// TIA Portal project "práctica 20_ comuniacion de plcs" (V15)

(* hardware
DEVICE "S7-1200 station_2"  S7-1200 Station
   slot 0: "Rack_0"  S7-1200 Rack  Rack  V1.0
   slot 1: "PLC_2"  CPU 1214C AC/DC/Rly  6ES7 214-1BG40-0XB0  V4.2
DEVICE "S7-1200 station_1"  S7-1200 Station
   slot 0: "Rack_0"  S7-1200 Rack  Rack  V1.0
   slot 1: "PLC_1"  CPU 1214C AC/DC/Rly  6ES7 214-1BG40-0XB0  V4.2
*)

// ===== PLC "PLC_1"  CPU 1214C AC/DC/Rly =====

VAR_GLOBAL   // PLC tag table "Tabla de variables estándar"
   "System_Byte" AT %MB253 : Byte;
   "FirstScan" AT %M253.0 : Bool;
   "DiagStatusUpdate" AT %M253.1 : Bool;
   "AlwaysTRUE" AT %M253.2 : Bool;
   "AlwaysFALSE" AT %M253.3 : Bool;
   "Clock_Byte" AT %MB254 : Byte;
   "Clock_10Hz" AT %M254.0 : Bool;
   "Clock_5Hz" AT %M254.1 : Bool;
   "Clock_2.5Hz" AT %M254.2 : Bool;
   "Clock_2Hz" AT %M254.3 : Bool;
   "Clock_1.25Hz" AT %M254.4 : Bool;
   "Clock_1Hz" AT %M254.5 : Bool;
   "Clock_0.625Hz" AT %M254.6 : Bool;
   "Clock_0.5Hz" AT %M254.7 : Bool;
   "info a enviar" AT %MW1 : Int;
END_VAR

// folder: System blocks/Program resources

DATA_BLOCK "IEC_Counter_0_DB"   // DB2
{ S7_Optimized_Access := 'TRUE' }
AUTHOR : Simatic
FAMILY : IEC
NAME : CNTR
VERSION : 1.0
// stored: InstanceOfName IEC_COUNTER
"IEC_COUNTER"
BEGIN
END_DATA_BLOCK

// folder: (top level)

ORGANIZATION_BLOCK "Main"   // OB1, LAD, ProgramCycle
TITLE = "Main Program Sweep (Cycle)"
{ S7_Optimized_Access := 'TRUE' }
VERSION : 0.1
   VAR_INPUT
      Initial_Call : Bool;   // Initial call of this OB
      Remanence : Bool;   // =True, if remanent data are available
   END_VAR
BEGIN

REGION Network 1
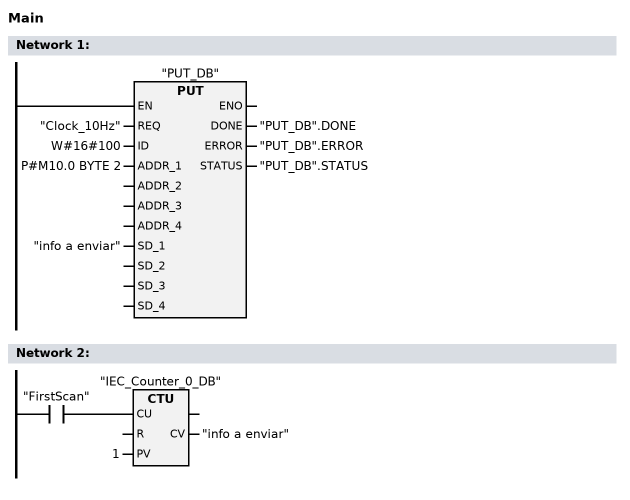
   "PUT_DB"(REQ := "Clock_10Hz",   // PUT
            ID := W#16#100,
            ADDR_1 := P#M10.0 BYTE 2,
            SD_1 := "info a enviar",
            DONE => "PUT_DB".DONE,
            ERROR => "PUT_DB".ERROR,
            STATUS => "PUT_DB".STATUS);
END_REGION

REGION Network 2
   "IEC_Counter_0_DB".CTU(CU := "FirstScan", PV := 1, CV => "info a enviar");
END_REGION
END_ORGANIZATION_BLOCK

// ===== PLC "PLC_2"  CPU 1214C AC/DC/Rly =====

VAR_GLOBAL   // PLC tag table "Tabla de variables estándar"
   "System_Byte" AT %MB253 : Byte;
   "FirstScan" AT %M253.0 : Bool;
   "DiagStatusUpdate" AT %M253.1 : Bool;
   "AlwaysTRUE" AT %M253.2 : Bool;
   "AlwaysFALSE" AT %M253.3 : Bool;
   "Clock_Byte" AT %MB254 : Byte;
   "Clock_10Hz" AT %M254.0 : Bool;
   "Clock_5Hz" AT %M254.1 : Bool;
   "Clock_2.5Hz" AT %M254.2 : Bool;
   "Clock_2Hz" AT %M254.3 : Bool;
   "Clock_1.25Hz" AT %M254.4 : Bool;
   "Clock_1Hz" AT %M254.5 : Bool;
   "Clock_0.625Hz" AT %M254.6 : Bool;
   "Clock_0.5Hz" AT %M254.7 : Bool;
   "info recibida" AT %MW10 : Int;
   "info traida" AT %MW5 : Int;
END_VAR

ORGANIZATION_BLOCK "Main"   // OB1, LAD, ProgramCycle
TITLE = "Main Program Sweep (Cycle)"
{ S7_Optimized_Access := 'TRUE' }
VERSION : 0.1
   VAR_INPUT
      Initial_Call : Bool;   // Initial call of this OB
      Remanence : Bool;   // =True, if remanent data are available
   END_VAR
BEGIN

REGION Network 1
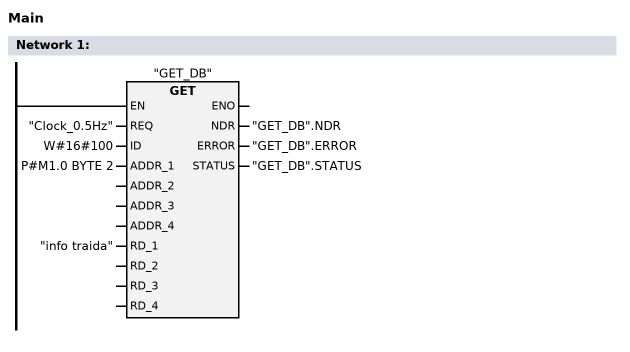
   "GET_DB"(REQ := "Clock_0.5Hz",   // GET
            ID := W#16#100,
            ADDR_1 := P#M1.0 BYTE 2,
            RD_1 := "info traida",
            NDR => "GET_DB".NDR,
            ERROR => "GET_DB".ERROR,
            STATUS => "GET_DB".STATUS);
END_REGION
END_ORGANIZATION_BLOCK